{attribute 'GeneratedUsingTerminal: AT2026-0250-0022'}
{attribute addProperty BoxType "AT2026-0250-0022"}
{attribute addProperty Id "A_0079_AT2002_5249_0018_AT2002_5249AT2002_33A3DF1B80"}
{attribute addProperty CRC "3211956198"}
{attribute addProperty Size "80"}
TYPE A_0067_AT2026_0250_0022_AT2026_0250_BF728FE6 EXTENDS AT2026_A7FEA1CF :
STRUCT
	{attribute addProperty Name "A_0079_AT2002_5249_0018_AT2002_5249"}
	{attribute addProperty PreviousPort "A_0067(AT2026-0250-0022) (AT2026-0250) : B"}
	A_0079_AT2002_5249_0018_AT2002_5249 : AT2002_33A3DF1B;
END_STRUCT
END_TYPE

(* stored: Version 1.2.0.0, ProductVersion 3.1.4024.9
   DUT A_0067_AT2026_0250_0022_AT2026_0250_BF728FE6: Id {ef39ce81-b2a7-4054-a333-15a9d0aaa07c} *)
